// TwinCAT 3 PLC project Untitled1
// ProgramVersion: 3.1.4024.0
// libraries:
//   Tc2_Standard, * (Beckhoff Automation GmbH)
//   Tc2_System, * (Beckhoff Automation GmbH)
//   Tc3_Module, * (Beckhoff Automation GmbH)
// project tree:
//   / PlcTask.TcTTO
//   POUs/ F_ReturnBitInDword.TcPOU, MAIN.TcPOU
// real-time tasks:
//   TASK PlcTask: cycle T#10ms, priority 20, ADS port 350

CONFIGURATION Untitled1
    RESOURCE PLC ON TwinCAT3
        TASK PlcTask(INTERVAL := T#10ms, PRIORITY := 20);
        PROGRAM MAIN WITH PlcTask : MAIN;
    END_RESOURCE
END_CONFIGURATION

// ---- POUs/MAIN.TcPOU
PROGRAM MAIN
VAR
	MyDword		: DWORD;
	ScannerIndex	: UINT;
	
	bitResult		: BOOL;
END_VAR


bitResult	:= F_ReturnBitInDword(inDword:= MyDword,inIndex:= ScannerIndex);

END_PROGRAM

// ---- POUs/F_ReturnBitInDword.TcPOU
FUNCTION F_ReturnBitInDword : BOOL
VAR_INPUT
	inDword		: DWORD;// The DWORD you wnat to inspect for bit level
	inIndex		: UINT;// Which bit in the DWORD do you want to know its level		
END_VAR
VAR
END_VAR

IF inIndex = 0 THEN
	F_ReturnBitInDword	:= inDword.0;
ELSIF inIndex = 1 THEN
	F_ReturnBitInDword	:= inDword.1;
ELSIF inIndex = 2 THEN
	F_ReturnBitInDword	:= inDword.2;
ELSIF inIndex = 3 THEN
	F_ReturnBitInDword	:= inDword.3;
ELSIF inIndex = 4 THEN
	F_ReturnBitInDword	:= inDword.4;
ELSIF inIndex = 5 THEN
	F_ReturnBitInDword	:= inDword.5;
ELSIF inIndex = 6 THEN
	F_ReturnBitInDword	:= inDword.6;
ELSIF inIndex = 7 THEN
	F_ReturnBitInDword	:= inDword.7;
ELSIF inIndex = 8 THEN
	F_ReturnBitInDword	:= inDword.8;
ELSIF inIndex = 9 THEN
	F_ReturnBitInDword	:= inDword.9;
ELSIF inIndex = 10 THEN
	F_ReturnBitInDword	:= inDword.10;
ELSIF inIndex = 11 THEN
	F_ReturnBitInDword	:= inDword.11;
ELSIF inIndex = 12 THEN
	F_ReturnBitInDword	:= inDword.12;
ELSIF inIndex = 13 THEN
	F_ReturnBitInDword	:= inDword.13;
ELSIF inIndex = 14 THEN
	F_ReturnBitInDword	:= inDword.14;
ELSIF inIndex = 15 THEN
	F_ReturnBitInDword	:= inDword.15;
ELSIF inIndex = 16 THEN
	F_ReturnBitInDword	:= inDword.16;
ELSIF inIndex = 17 THEN
	F_ReturnBitInDword	:= inDword.17;
ELSIF inIndex = 18 THEN
	F_ReturnBitInDword	:= inDword.18;
ELSIF inIndex = 19 THEN
	F_ReturnBitInDword	:= inDword.19;
ELSIF inIndex = 20 THEN
	F_ReturnBitInDword	:= inDword.20;
ELSIF inIndex = 21 THEN
	F_ReturnBitInDword	:= inDword.21;
ELSIF inIndex = 22 THEN
	F_ReturnBitInDword	:= inDword.22;
ELSIF inIndex = 23 THEN
	F_ReturnBitInDword	:= inDword.23;
ELSIF inIndex = 24 THEN
	F_ReturnBitInDword	:= inDword.24;
ELSIF inIndex = 25 THEN
	F_ReturnBitInDword	:= inDword.25;
ELSIF inIndex = 26 THEN
	F_ReturnBitInDword	:= inDword.26;
ELSIF inIndex = 27 THEN
	F_ReturnBitInDword	:= inDword.27;
ELSIF inIndex = 28 THEN
	F_ReturnBitInDword	:= inDword.28;
ELSIF inIndex = 29 THEN
	F_ReturnBitInDword	:= inDword.29;
ELSIF inIndex = 30 THEN
	F_ReturnBitInDword	:= inDword.30;
ELSIF inIndex = 31 THEN
	F_ReturnBitInDword	:= inDword.31;
ELSE
	F_ReturnBitInDword:= TRUE;
END_IF

END_FUNCTION
